FUNCTION_BLOCK CM_AO_V2
VAR_INPUT
	IN_ON : BOOL;

	PI_PV : DINT; // Input from sensor or other device which should control
	
	SP_AUTO : DINT;
	SP_MAN: DINT;
	
	PI_HMI_HAND_ON :BOOL;
	
	
	Local_MODE_request : ENUM_MODE_HANDLER;
	Global_MODE_request : ENUM_MODE_HANDLER;
	
	
	//PID_PARAMS : ST_CTRL_PID_PARAMS;
	
	
	//ALARMS:
	PI_AlarmHighHighEnable : BOOL;
	PI_AlarmHighEnable : BOOL;
	PI_AlarmLowEnable : BOOL;
	PI_AlarmLowLowEnable : BOOL;
	
	PI_AlarmHighHighLimit : REAL;
	PI_AlarmHighLimit : REAL;
	PI_AlarmLowLimit : REAL;
	PI_AlarmLowLowLimit : REAL;
	
	PI_AlarmDelay_HH : LREAL;
	PI_AlarmDelay_H : LREAL;
	PI_AlarmDelay_L : LREAL;
	PI_AlarmDelay_LL : LREAL;
	
	Alarm_Ack_HH : BOOL;
	Alarm_Ack_H : BOOL;
	Alarm_Ack_L : BOOL;
	Alarm_Ack_LL : BOOL;
	
	PI_Interlock : BOOL;
	
	ENABLE_SCALING : BOOL;
	PI_PV_MAX_IN : INT;
	PI_PV_MIN_IN : INT;
	PI_PV_MAX_OUT : INT;
	PI_PV_MIN_OUT : INT;
END_VAR
VAR_OUTPUT
	
	PO_AUTO_ON :BOOL;
	PO_MANUAL_ON : BOOL;
	PO_HMI_HAND_ON : BOOL;
	
	PO_OUT_ON : BOOL;
	PO_OUT_OFF :BOOL;
	
	PO_Interlocked : BOOL;
	
	PO_PV_SCALED : REAL;
	
	PO_ALARM_HH : BOOL;
	PO_ALARM_H : BOOL;
	PO_ALARM_L : BOOL;
	PO_ALARM_LL : BOOL;
END_VAR
VAR_IN_OUT
	
END_VAR
VAR
	SR_Auto: SR;
	SR_Manual : SR;
	
	Alarm_limit_Exceeded_HH : BOOL;
	Alarm_limit_Exceeded_H : BOOL;
	Alarm_limit_Exceeded_L : BOOL;
	Alarm_limit_Exceeded_LL : BOOL;
	
	alarmDelay_HH : systemTimeDelay;
	alarmDelay_H : systemTimeDelay;
	alarmDelay_L : systemTimeDelay;
	alarmDelay_LL : systemTimeDelay;
	
	DelayForHistorianBit_HH: TON;
	DelayForHistorianBit_H: TON;
	DelayForHistorianBit_L: TON;
	DelayForHistorianBit_LL: TON;
	
	HistorianBit_HH :BOOL;
	HistorianBit_H :BOOL;
	HistorianBit_L :BOOL;
	HistorianBit_LL :BOOL;
	
	MODE_HANDLER : FB_MODE_HANDLER;
	
	scale : Tc2_ControllerToolbox.FB_CTRL_SCALE;
	scaleParams : ST_CTRL_SCALE_PARAMS;
	
	MODEHANDLER_AUTO_ON : BOOL;
	MODEHANDLER_MANUAL_ON : BOOL;
END_VAR

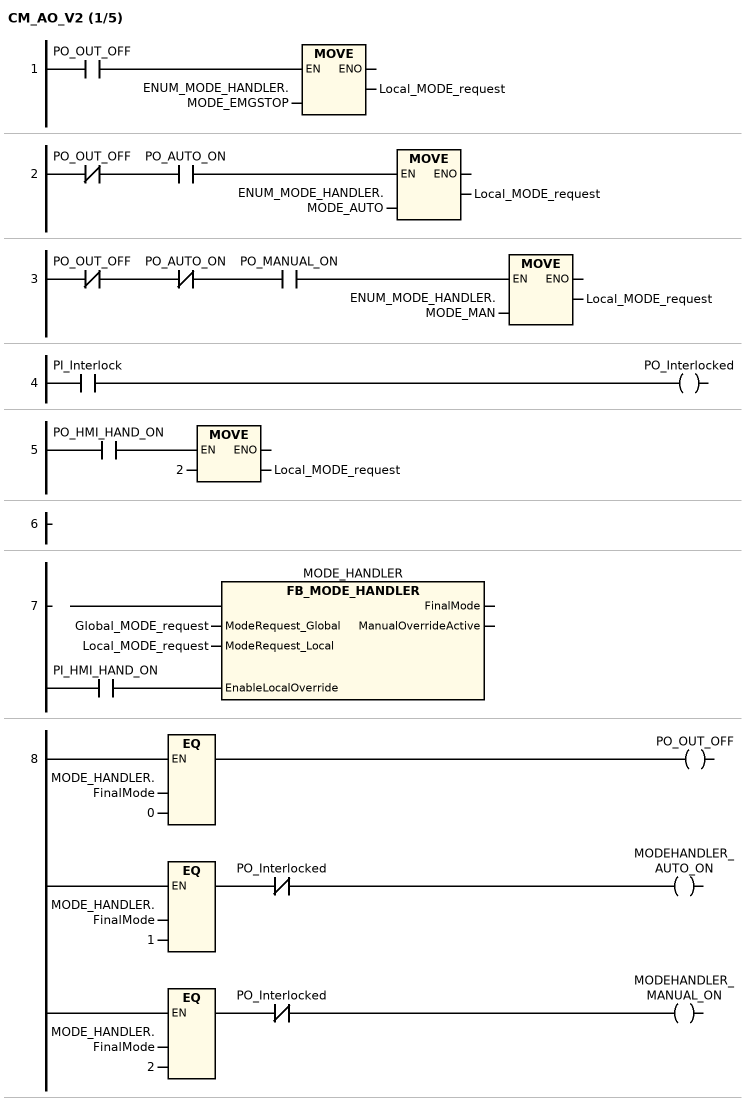
// NETWORK 1
IF PO_OUT_OFF THEN Local_MODE_request := ENUM_MODE_HANDLER.MODE_EMGSTOP; END_IF

// NETWORK 2
IF NOT PO_OUT_OFF AND PO_AUTO_ON THEN Local_MODE_request := ENUM_MODE_HANDLER.MODE_AUTO; END_IF

// NETWORK 3
IF NOT PO_OUT_OFF AND NOT PO_AUTO_ON AND PO_MANUAL_ON THEN Local_MODE_request := ENUM_MODE_HANDLER.MODE_MAN; END_IF

// NETWORK 4
PO_Interlocked := PI_Interlock;

// NETWORK 5
IF PO_HMI_HAND_ON THEN Local_MODE_request := 2; END_IF

// NETWORK 6

// NETWORK 7
MODE_HANDLER(
    ModeRequest_Global := Global_MODE_request,
    ModeRequest_Local := Local_MODE_request,
    EnableLocalOverride := PI_HMI_HAND_ON); // FB_MODE_HANDLER

// NETWORK 8
PO_OUT_OFF := MODE_HANDLER.FinalMode = 0;
MODEHANDLER_AUTO_ON := MODE_HANDLER.FinalMode = 1 AND NOT PO_Interlocked;
MODEHANDLER_MANUAL_ON := MODE_HANDLER.FinalMode = 2 AND NOT PO_Interlocked;

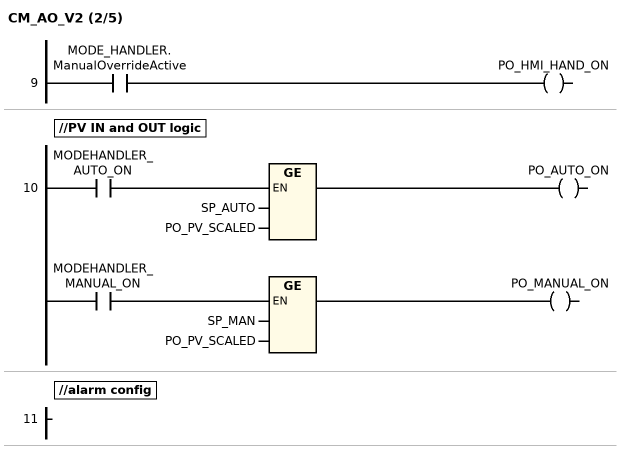
// NETWORK 9
PO_HMI_HAND_ON := MODE_HANDLER.ManualOverrideActive;

// NETWORK 10
// label: //PV IN and OUT logic
PO_AUTO_ON := MODEHANDLER_AUTO_ON AND SP_AUTO >= PO_PV_SCALED;
PO_MANUAL_ON := MODEHANDLER_MANUAL_ON AND SP_MAN >= PO_PV_SCALED;

// NETWORK 11
// label: //alarm config

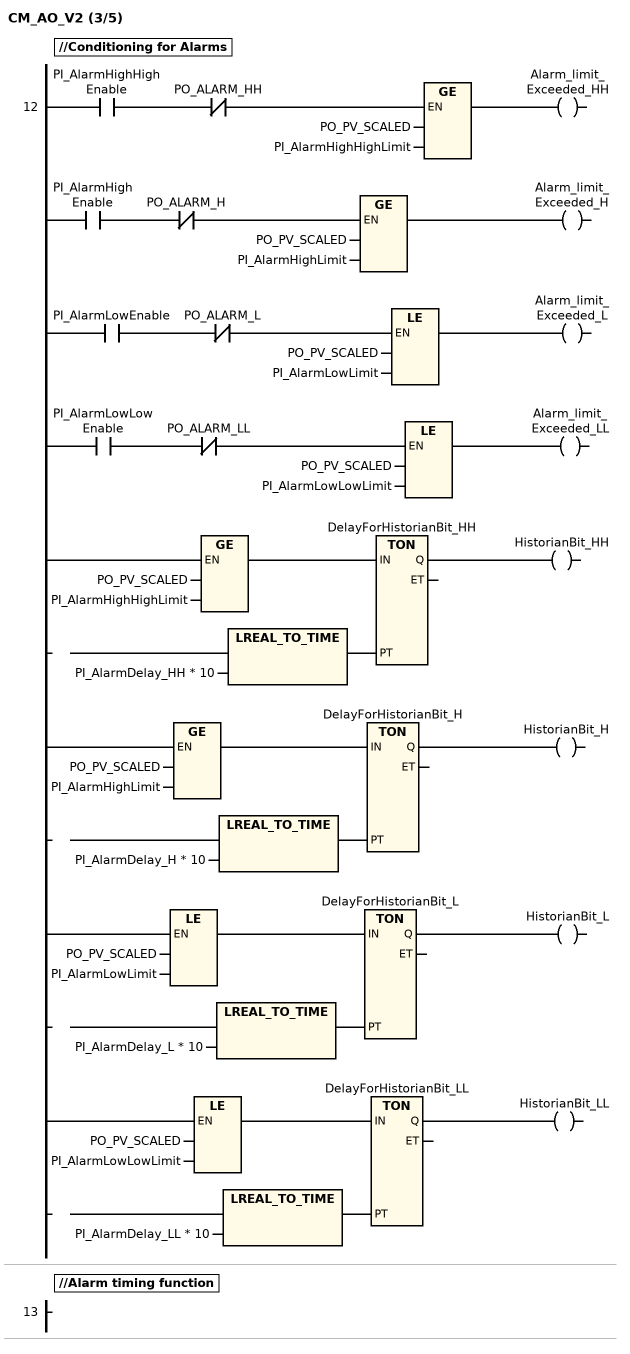
// NETWORK 12
// label: //Conditioning for Alarms
Alarm_limit_Exceeded_HH := PI_AlarmHighHighEnable AND NOT PO_ALARM_HH AND PO_PV_SCALED >= PI_AlarmHighHighLimit;
Alarm_limit_Exceeded_H := PI_AlarmHighEnable AND NOT PO_ALARM_H AND PO_PV_SCALED >= PI_AlarmHighLimit;
Alarm_limit_Exceeded_L := PI_AlarmLowEnable AND NOT PO_ALARM_L AND PO_PV_SCALED <= PI_AlarmLowLimit;
Alarm_limit_Exceeded_LL := PI_AlarmLowLowEnable AND NOT PO_ALARM_LL AND PO_PV_SCALED <= PI_AlarmLowLowLimit;
DelayForHistorianBit_HH(IN := PO_PV_SCALED >= PI_AlarmHighHighLimit, PT := LREAL_TO_TIME(PI_AlarmDelay_HH * 10)); // TON
HistorianBit_HH := DelayForHistorianBit_HH.Q;
DelayForHistorianBit_H(IN := PO_PV_SCALED >= PI_AlarmHighLimit, PT := LREAL_TO_TIME(PI_AlarmDelay_H * 10)); // TON
HistorianBit_H := DelayForHistorianBit_H.Q;
DelayForHistorianBit_L(IN := PO_PV_SCALED <= PI_AlarmLowLimit, PT := LREAL_TO_TIME(PI_AlarmDelay_L * 10)); // TON
HistorianBit_L := DelayForHistorianBit_L.Q;
DelayForHistorianBit_LL(IN := PO_PV_SCALED <= PI_AlarmLowLowLimit, PT := LREAL_TO_TIME(PI_AlarmDelay_LL * 10)); // TON
HistorianBit_LL := DelayForHistorianBit_LL.Q;

// NETWORK 13
// label: //Alarm timing function

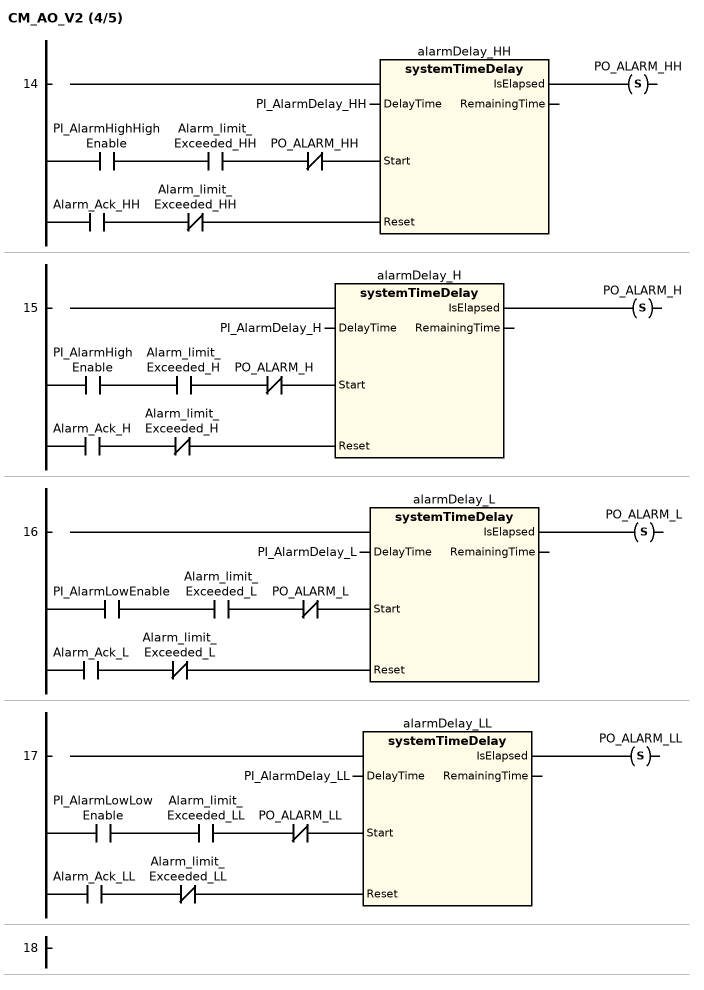
// NETWORK 14
alarmDelay_HH(
    DelayTime := PI_AlarmDelay_HH,
    Start := PI_AlarmHighHighEnable AND Alarm_limit_Exceeded_HH AND NOT PO_ALARM_HH,
    Reset := Alarm_Ack_HH AND NOT Alarm_limit_Exceeded_HH); // systemTimeDelay
PO_ALARM_HH S= alarmDelay_HH.IsElapsed;

// NETWORK 15
alarmDelay_H(
    DelayTime := PI_AlarmDelay_H,
    Start := PI_AlarmHighEnable AND Alarm_limit_Exceeded_H AND NOT PO_ALARM_H,
    Reset := Alarm_Ack_H AND NOT Alarm_limit_Exceeded_H); // systemTimeDelay
PO_ALARM_H S= alarmDelay_H.IsElapsed;

// NETWORK 16
alarmDelay_L(
    DelayTime := PI_AlarmDelay_L,
    Start := PI_AlarmLowEnable AND Alarm_limit_Exceeded_L AND NOT PO_ALARM_L,
    Reset := Alarm_Ack_L AND NOT Alarm_limit_Exceeded_L); // systemTimeDelay
PO_ALARM_L S= alarmDelay_L.IsElapsed;

// NETWORK 17
alarmDelay_LL(
    DelayTime := PI_AlarmDelay_LL,
    Start := PI_AlarmLowLowEnable AND Alarm_limit_Exceeded_LL AND NOT PO_ALARM_LL,
    Reset := Alarm_Ack_LL AND NOT Alarm_limit_Exceeded_LL); // systemTimeDelay
PO_ALARM_LL S= alarmDelay_LL.IsElapsed;

// NETWORK 18

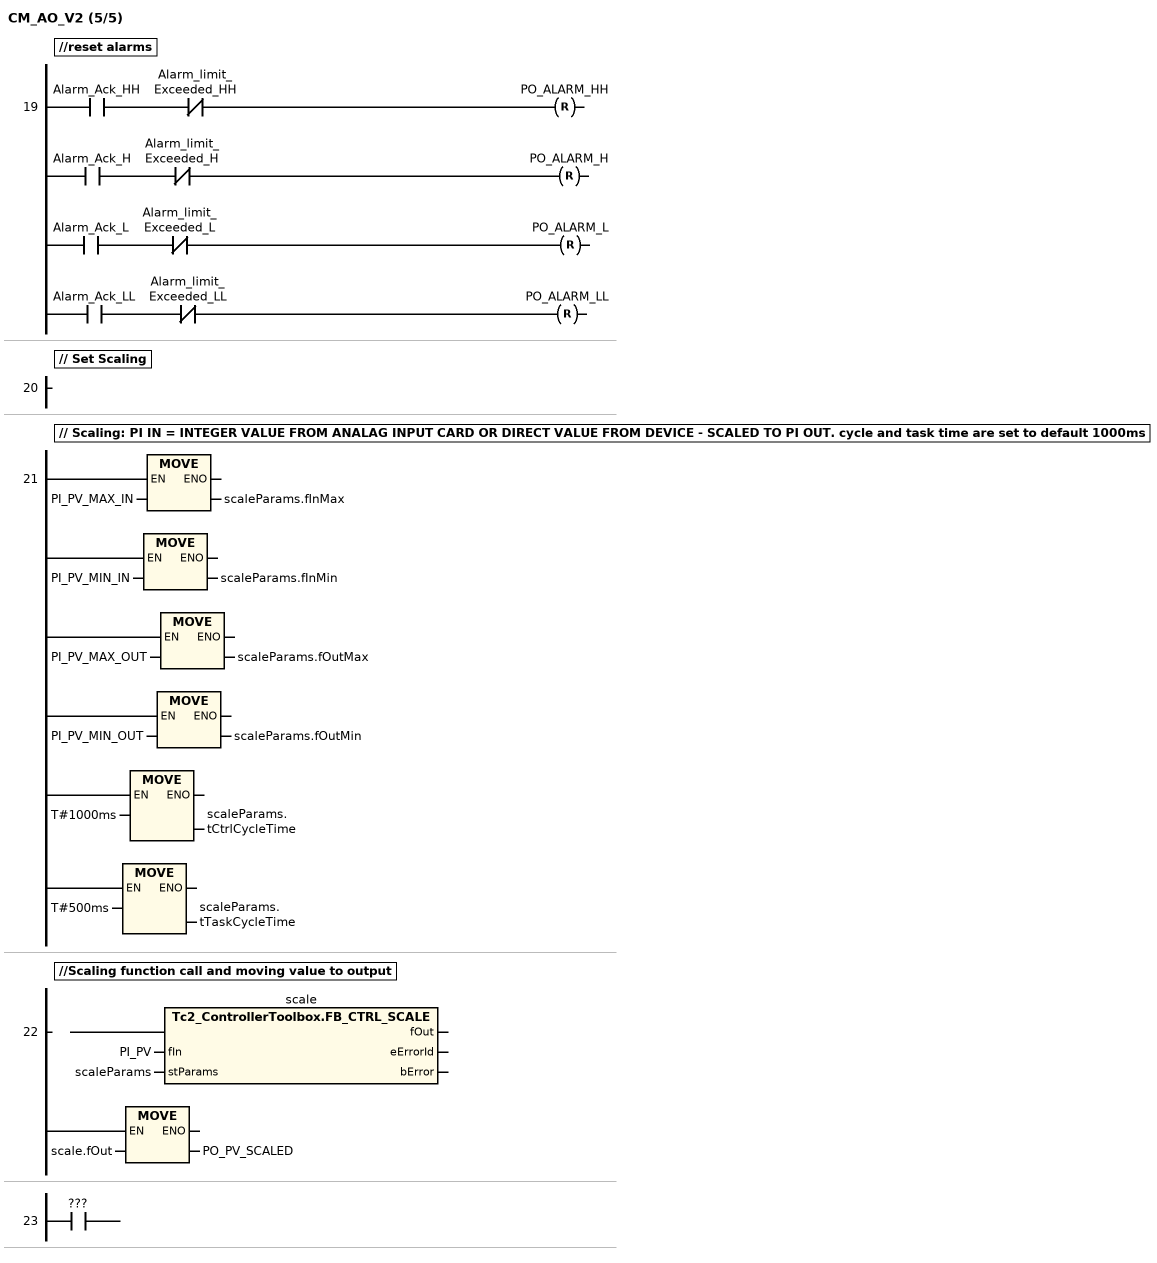
// NETWORK 19
// label: //reset alarms
PO_ALARM_HH R= Alarm_Ack_HH AND NOT Alarm_limit_Exceeded_HH;
PO_ALARM_H R= Alarm_Ack_H AND NOT Alarm_limit_Exceeded_H;
PO_ALARM_L R= Alarm_Ack_L AND NOT Alarm_limit_Exceeded_L;
PO_ALARM_LL R= Alarm_Ack_LL AND NOT Alarm_limit_Exceeded_LL;

// NETWORK 20
// label: // Set Scaling

// NETWORK 21
// label: // Scaling: PI IN = INTEGER VALUE FROM ANALAG INPUT CARD OR DIRECT VALUE FROM DEVICE - SCALED TO PI OUT. cycle and task time are set to default 1000ms
scaleParams.fInMax := PI_PV_MAX_IN;
scaleParams.fInMin := PI_PV_MIN_IN;
scaleParams.fOutMax := PI_PV_MAX_OUT;
scaleParams.fOutMin := PI_PV_MIN_OUT;
scaleParams.tCtrlCycleTime := T#1000ms;
scaleParams.tTaskCycleTime := T#500ms;

// NETWORK 22
// label: //Scaling function call and moving value to output
scale(fIn := PI_PV, stParams := scaleParams); // Tc2_ControllerToolbox.FB_CTRL_SCALE
PO_PV_SCALED := scale.fOut;

// NETWORK 23

END_FUNCTION_BLOCK

(* stored: Version 1.1.0.1, ProductVersion 3.1.4024.13
   POU CM_AO_V2: Id {eb4da971-634c-41e8-879f-dfb9f5d3ec38}, SpecialFunc None *)
